FUNCTION_BLOCK FB_UR5 EXTENDS FB_ROB_MANIP IMPLEMENTS ITF_BA_6Axis, ITF_CommunicationModul
VAR_INPUT
END_VAR
VAR_OUTPUT
END_VAR
VAR
	PiNPl: Skill_PickPlace;
END_VAR

StateMachine();


//Reference to Skills
PiNPl(Rob:=ADR(THIS^));

//ComConfig

ComConfig.sIPAddress:='127.0.0.1';
ComConfig.nPort:= 5432;

METHOD Connect : BOOL
VAR_INPUT
END_VAR
END_METHOD

PROPERTY Connected : BOOL
GET
END_GET
END_PROPERTY

METHOD Disconnect : BOOL
VAR_INPUT
END_VAR
END_METHOD

{warning 'Add method implementation '}
METHOD MC_MoveAxesRelative : BOOL
VAR_INPUT
	axes	: ARRAY [1..6] OF FB_Axis;
	offsets	: ARRAY [1..6] OF REAL;
END_VAR
END_METHOD

{warning 'Add method implementation '}
METHOD MC_MoveJ : BOOL
VAR_INPUT
	target	: stTarget3D;
END_VAR
IF _state=eState.Active THEN
// 	P_TargetReached:=FALSE;
END_IF
END_METHOD

{warning 'Add method implementation '}
METHOD MC_MoveL : BOOL
VAR_INPUT
	target	: stTarget3D;
END_VAR
END_METHOD

{warning 'Add method implementation '}
METHOD MC_ReadActualVelocity : stPose
END_METHOD

{warning 'Add method implementation '}
METHOD MC_ReadAnalogInput : LREAL
VAR_INPUT
	input	: INT;
END_VAR
END_METHOD

{warning 'Add method implementation '}
METHOD MC_ReadDigitalInput : BOOL
VAR_INPUT
	input	: INT;
END_VAR
END_METHOD

{warning 'Add method implementation '}
METHOD MC_SetDigitalOutput : BOOL
VAR_INPUT
	output	: INT;
	value	: BOOL;
END_VAR
END_METHOD

{warning 'Add method implementation '}
METHOD MC_SetOperationMode : BOOL
VAR_INPUT
	mode	: eMode;
END_VAR
_mode:=mode;
END_METHOD

METHOD MC_SpeedOverride : INT
VAR_INPUT
	factor: REAL;
END_VAR
END_METHOD

METHOD onActivate : BOOL
// ---- Init ----
transitionresult:=eResult.None;



// ---- Change ----

// _mode:= eMode.Automatic;




// ---- Check ----
transitionresult := eResult.SUCCESS;


// ---- Change State ----
IF transitionresult= eResult.SUCCESS THEN
	State:=eState.Active;
ELSIF transitionresult= eResult.FAILURE THEN
	State:=eState.Inactive;
ELSIF transitionresult= eResult.ERROR THEN
	State:=eState.ErrorProcessing;
ELSE
	ADSLOGSTR(ADSLOG_MSGTYPE_WARN,'Transitionresult from onActivate is None','');
END_IF
END_METHOD

METHOD onCleanup : BOOL
// ---- Init ----
transitionresult:=eResult.None;



// ---- Change ----

_mode:= eMode.Manual;




// ---- Check ----
transitionresult := eResult.SUCCESS;


// ---- Change State ----
IF transitionresult= eResult.SUCCESS THEN
	State:=eState.Unconfigured;
ELSIF transitionresult= eResult.FAILURE THEN
	ADSLOGSTR(ADSLOG_MSGTYPE_WARN,'Transitionresult from onCleanup is FAILURE ','');
ELSIF transitionresult= eResult.ERROR THEN
	State:=eState.ErrorProcessing;
ELSE
	ADSLOGSTR(ADSLOG_MSGTYPE_WARN,'Transitionresult from onCleanup is NONE','');
END_IF
END_METHOD

METHOD onConfigure : BOOL
// ---- Init ----
transitionresult:=eResult.None;



// ---- Change ----

_mode:= eMode.Manual;




// ---- Check ----
transitionresult := eResult.SUCCESS;


// ---- Change State ----
IF transitionresult= eResult.SUCCESS THEN
	State:=eState.Inactive;
ELSIF transitionresult= eResult.FAILURE THEN
	State:=eState.Unconfigured;
ELSIF transitionresult= eResult.ERROR THEN
	State:=eState.ErrorProcessing;
ELSE
	ADSLOGSTR(ADSLOG_MSGTYPE_WARN,'Transitionresult from onConfigure is None','');
END_IF
END_METHOD

METHOD onDeactivate : BOOL
// ---- Init ----
transitionresult:=eResult.None;



// ---- Change ----

_mode:= eMode.Manual;




// ---- Check ----
transitionresult := eResult.SUCCESS;


// ---- Change State ----
IF transitionresult= eResult.SUCCESS THEN
	State:=eState.Inactive;
ELSIF transitionresult= eResult.FAILURE THEN
	ADSLOGSTR(ADSLOG_MSGTYPE_WARN,'Transitionresult from onDeactivate is FAILURE','');
ELSIF transitionresult= eResult.ERROR THEN
	State:=eState.ErrorProcessing;
ELSE
	ADSLOGSTR(ADSLOG_MSGTYPE_WARN,'Transitionresult from onDeactivate is None','');
END_IF
END_METHOD

METHOD onError : BOOL
// ---- Init ----
transitionresult:=eResult.None;



// ---- Change ----

_mode:= eMode.Manual;




// ---- Check ----
transitionresult := eResult.SUCCESS;


// ---- Change State ----
IF transitionresult= eResult.SUCCESS THEN
	State:=eState.Unconfigured;
ELSIF transitionresult= eResult.FAILURE THEN
	State:=eState.Finalized;
ELSIF transitionresult= eResult.ERROR THEN
	ADSLOGSTR(ADSLOG_MSGTYPE_WARN,'Transitionresult from onError is Error','');
ELSE
	ADSLOGSTR(ADSLOG_MSGTYPE_WARN,'Transitionresult from onError is None','');
END_IF
END_METHOD

METHOD onShutdown : BOOL
// ---- Init ----
transitionresult:=eResult.None;



// ---- Change ----

_mode:= eMode.Manual;




// ---- Check ----
transitionresult := eResult.SUCCESS;


// ---- Change State ----
IF transitionresult= eResult.SUCCESS THEN
	State:=eState.Finalized;
ELSIF transitionresult= eResult.FAILURE THEN
	ADSLOGSTR(ADSLOG_MSGTYPE_WARN,'Transitionresult from onShutdown is FAILURE','');
ELSIF transitionresult= eResult.ERROR THEN
	State:=eState.ErrorProcessing;
ELSE
	ADSLOGSTR(ADSLOG_MSGTYPE_WARN,'Transitionresult from onShutdown is None','');
END_IF
END_METHOD

METHOD ResetConnection : BOOL
VAR_INPUT
END_VAR
END_METHOD

END_FUNCTION_BLOCK

(* stored: Version 1.1.0.1, ProductVersion 3.1.4026.18
   POU FB_UR5: Id {7138b06d-6984-4953-8124-68042278758b}, SpecialFunc None
   Folder Communication: Id {962090cd-82cb-4129-9347-c8ac07fb90f4}
   Folder MotionControl: Id {9ed28985-c54d-42fa-8d69-76777d28de96}
   Folder StateControl: Id {da6218f9-6bd6-462f-bf56-7f509f8b869c}
   Method Connect: Id {ea0b7a54-6a8f-44d8-8b6a-a3c96ae90503}
   Property Connected: Id {37ba7a67-b4ee-42b5-aea8-1f3fba5d5175}
   Get Get: Id {d4b74009-4a4c-4abb-b825-78ae2fd94b8a}
   Method Disconnect: Id {81d53a8c-a37e-4c7e-ab45-5d8abfba1924}
   Method MC_MoveAxesRelative: Id {dc6eaf0b-bda4-4a71-9f22-4f43caa591cf}
   Method MC_MoveJ: Id {e4cbbe25-0003-4a3a-941f-ba8ea400b2d6}
   Method MC_MoveL: Id {fac605cc-f9e9-41e9-8d84-7a37c1c2f07e}
   Method MC_ReadActualVelocity: Id {8fcd44ac-c416-4fa2-be4a-a96c08398ed8}
   Method MC_ReadAnalogInput: Id {f3e9cd2c-1bdb-4b96-8862-1b49b481f6f5}
   Method MC_ReadDigitalInput: Id {fa482187-c1ce-433f-9f9a-2cc320aaca90}
   Method MC_SetDigitalOutput: Id {9228931f-d00e-488b-96fa-facc797720c5}
   Method MC_SetOperationMode: Id {b77d92d3-2c73-432f-b915-482766ea505a}
   Method MC_SpeedOverride: Id {b4de7407-a668-4de0-9ba6-a503ff62da73}
   Method onActivate: Id {dc70c063-7d50-424b-ae24-a3b2e8b82a59}
   Method onCleanup: Id {c5444503-9fdd-4b71-a65c-fd5cddb6bb43}
   Method onConfigure: Id {89188265-a853-4cc7-b2e5-efc6c3414bec}
   Method onDeactivate: Id {b48ff0b4-7768-470e-ba5f-bd75733f4dc6}
   Method onError: Id {40b32895-142b-4a04-aa6c-109bbaa0fa6c}
   Method onShutdown: Id {5ad9cf95-ea02-430b-a003-aed2972e9fe8}
   Method ResetConnection: Id {ab760c43-0912-46a9-8200-3ef0d14f05e9} *)
